Omron CX-Programmer project NewProject (CX-Programmer 9.75)

# PLC AUTODOOR_PROJECT: CJ2M CPU11

## Global symbols (name address type ; comment)
0.00 BOOL  ; IR SENSOR
0.01 BOOL  ; LS1
0.02 BOOL  ; LS2
0.03 BOOL  ; LS3
100.00 BOOL  ; MOTOR
100.01 BOOL  ; MOTOR REV
T0000 BOOL  ; T0

## Program NewProgram1 (cyclic task 0)

### Section Section1

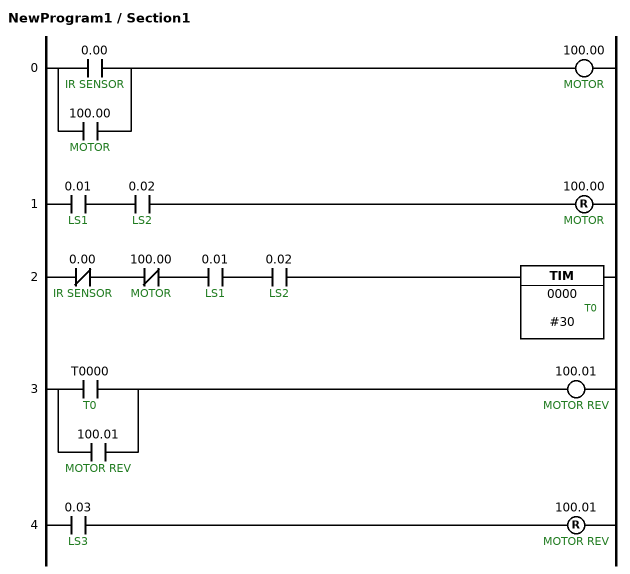
; rung 0
LD 0.00  ; IR SENSOR
OR 100.00  ; MOTOR
OUT 100.00  ; MOTOR
; rung 1
LD 0.01  ; LS1
AND 0.02  ; LS2
RSET 100.00  ; MOTOR
; rung 2
LDNOT 0.00  ; IR SENSOR
ANDNOT 100.00  ; MOTOR
AND 0.01  ; LS1
AND 0.02  ; LS2
TIM 0000 #30  ; T0
; rung 3
LD T0000  ; T0
OR 100.01  ; MOTOR REV
OUT 100.01  ; MOTOR REV
; rung 4
LD 0.03  ; LS3
RSET 100.01  ; MOTOR REV

### Section END
; rung 0
END(001)